# EPICS substitutions: respmat/respmatApp/Db/userHost.substitutions
# Example substitutions file

file "db/dbExample1.db" {
    { user = "lyyangHost" }
}

file db/dbExample2.db {
    pattern { user, no, scan }
        { "lyyangHost", 1, "1 second" }
        { "lyyangHost", 2, "2 second" }
        { "lyyangHost", 3, "5 second" }
}
